// TIA Portal V17 export
// export: Created 2024-01-30T08:49:17.0979588Z, ExportSetting WithDefaults, DisplayName Totally Integrated Automation Portal, DisplayVersion V17 Update 6, DisplayName TIA Portal Openness, DisplayVersion V17 Update 6, DisplayName TIA Portal Version Control Interface, DisplayVersion V17, DisplayName STEP 7 Professional, DisplayVersion V17 Update 6, DisplayName STEP 7 Safety, DisplayVersion V17 Update 6, DisplayName WinCC Advanced, DisplayVersion V17 Update 6
TYPE "OvenTemperature"
// stored: IsFailsafeCompliant false
   STRUCT
      Temperature_1 : Real := 1.0;
      Temperature_2 : Real := 4.0;
      Temperature_3 : Real := 16.0;
      "Time" : LDT;
   END_STRUCT;
END_TYPE
